// TIA Portal project "GestionCMD" (V17)

(* hardware
DEVICE "S7-1500/ET200MP station_1"  S7-1500 station
   slot 0: "Rail_0"  Rack  6ES7 590-1***0-0AA0
   slot 1: "PLC_1"  CPU 1516-3 PN/DP  6ES7 516-3AN02-0AB0  V2.9
      slot 3: "CPU display_1"  6ES7591-1BA00-0AA0
      slot 32768: "PROFINET interface_1"  X1
         slot 32769: "Port_1"  X1 P1
         slot 32770: "Port_2"  X1 P2
      slot 33024: "PROFINET interface_2"  X2
         slot 33025: "Port_1"  X2 P1
      slot 33280: "DP interface_1"  X3
      slot 34817: "Virtual CP interface port_1"  Virtual CP interface port  Virtual CP interface port
DEVICE "HMI_1"  KTP400 Comfort
   slot 0: "HMI_1"  KTP400 Comfort  6AV2 124-2DC01-0AX0  17.0.0.0
   slot 1: "HMI_RT_1"  KTP400 Comfort  6AV2 124-2DC01-0AX0  17.0.0.0
   slot 5: "HMI_1.IE_CP_1"  PROFINET Interface  17.0.0.0
      slot 1: "PROFINET Interface_1"  PROFINET Interface
         slot 1: "Port_1"  Port
   slot 7: "HMI_1.MPI/DP_CP_1"  MPI/DP Interface  17.0.0.0
*)

// ===== PLC "PLC_1"  CPU 1516-3 PN/DP =====

VAR_GLOBAL   // PLC tag table "Default tag table"
   "Etape1" AT %M0.0 : Bool;
   "Etape2" AT %M0.1 : Bool;
   "Etape3" AT %M0.2 : Bool;
   "MonterBarriere" AT %Q0.0 : Bool;
   "DescenteBarriere" AT %Q0.1 : Bool;
   "VoiturePasser" AT %M0.3 : Bool;
   "N_fois_badge" AT %MW10 : Int;
   "PositionBasBarriere" AT %M2.0 : Bool;
   "SignalBadge" AT %M2.1 : Bool;
   "Tag_1" AT %Q0.2 : Bool;
   "UpLevel" AT %I0.0 : Bool;
   "DownLevel" AT %I0.1 : Bool;
   "LevelFC" AT %MW30 : Int;
   "LevelFB" AT %MW34 : Int;
   "Tag_2" AT %M4.0 : Bool;
   "Tag_3" AT %M4.1 : Bool;
   "Tag_4" AT %M4.2 : Bool;
   "Tag_5" AT %M4.3 : Bool;
   "trigger" AT %M4.4 : Bool;
END_VAR

DATA_BLOCK "FB1"   // DB3
{ S7_Optimized_Access := 'TRUE' }
VERSION : 0.1
// stored: InstanceOfName Block_1
"Block_1"
BEGIN
END_DATA_BLOCK

DATA_BLOCK "FillingFB_DB"   // DB4
{ S7_Optimized_Access := 'TRUE' }
VERSION : 0.1
// stored: InstanceOfName FillingFB
"FillingFB"
BEGIN
END_DATA_BLOCK

FUNCTION_BLOCK "Block_1"   // FB1, SCL
{ S7_Optimized_Access := 'TRUE' }
VERSION : 0.1
   VAR
      MyNBBadge : Int;
   END_VAR
BEGIN
   IF "Etape1" AND "N_fois_badge" <> 0 THEN
       "Etape2" := TRUE;
       "Etape1" := FALSE;
   END_IF;

   IF "Etape2" AND "VoiturePasser" <> 0 THEN
       "Etape3" := TRUE;
       "Etape2" := FALSE;
   END_IF;

   IF "Etape3" AND "PositionBasBarriere" <> 0 THEN
       "Etape1" := TRUE;
       "Etape3" := FALSE;
   END_IF;

   "R_TRIG_DB"(CLK:="SignalBadge");
   "F_Etape1"(CLK := "Etape1");

   IF "R_TRIG_DB".Q THEN
       "N_fois_badge" += 1;
   END_IF;

   IF "F_Etape1".Q THEN
       "N_fois_badge" -= 1;
   END_IF;

   #MyNBBadge := "N_fois_badge";
END_FUNCTION_BLOCK

FUNCTION_BLOCK "FillingFB"   // FB2, LAD
{ S7_Optimized_Access := 'TRUE' }
VERSION : 0.1
   VAR_INPUT
      uplevel : Bool;
      downlevel : Bool;
   END_VAR
   VAR_OUTPUT
      OutLevel : Int;
   END_VAR
   VAR
      volum : Int;
   END_VAR
BEGIN

REGION Network 2
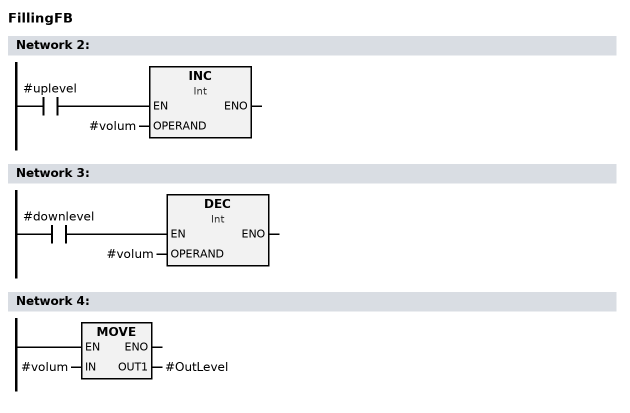
   RUNG wire#powerrail
      Contact( #uplevel )
      { S7_Templates := "DestType := Int" } Inc( #volum )
   END_RUNG
   // the same network as SCL:
   IF #uplevel THEN #volum := #volum + 1; END_IF;
END_REGION

REGION Network 3
   RUNG wire#powerrail
      Contact( #downlevel )
      { S7_Templates := "DestType := Int" } Dec( #volum )
   END_RUNG
   // the same network as SCL:
   IF #downlevel THEN #volum := #volum - 1; END_IF;
END_REGION

REGION Network 4
   RUNG wire#powerrail
      Move(in := #volum, out1 => #OutLevel)
   END_RUNG
   // the same network as SCL:
   #OutLevel := #volum;
END_REGION
END_FUNCTION_BLOCK

FUNCTION "FillingFC" : Void   // FC1, LAD
{ S7_Optimized_Access := 'TRUE' }
VERSION : 0.1
   VAR_INPUT
      uplevel : Bool;
      downlevel : Bool;
   END_VAR
   VAR_OUTPUT
      OutLevel : Int;
   END_VAR
   VAR_TEMP
      Volum : Int;
   END_VAR
   VAR CONSTANT
      Constant_1 : Int;
   END_VAR
BEGIN

REGION Network 1
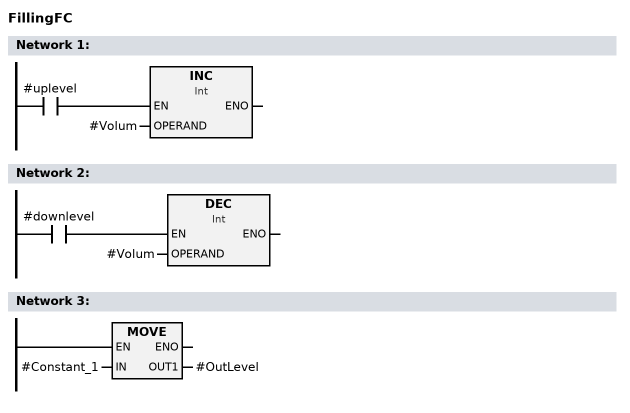
   RUNG wire#powerrail
      Contact( #uplevel )
      { S7_Templates := "DestType := Int" } Inc( #Volum )
   END_RUNG
   // the same network as SCL:
   IF #uplevel THEN #Volum := #Volum + 1; END_IF;
END_REGION

REGION Network 2
   RUNG wire#powerrail
      Contact( #downlevel )
      { S7_Templates := "DestType := Int" } Dec( #Volum )
   END_RUNG
   // the same network as SCL:
   IF #downlevel THEN #Volum := #Volum - 1; END_IF;
END_REGION

REGION Network 3
   RUNG wire#powerrail
      Move(in := #Constant_1, out1 => #OutLevel)
   END_RUNG
   // the same network as SCL:
   #OutLevel := #Constant_1;
END_REGION
END_FUNCTION

ORGANIZATION_BLOCK "Main"   // OB1, LAD, ProgramCycle
TITLE = "Main Program Sweep (Cycle)"
{ S7_Optimized_Access := 'TRUE' }
VERSION : 0.1
   VAR_INPUT
      Initial_Call : Bool;   // Initial call of this OB
      Remanence : Bool;   // =True, if remanent data are available
   END_VAR
   VAR_TEMP   // added for the SCL form of the ladder/FBD networks
      _w1 : Bool;
      _w2 : Bool;
   END_VAR
BEGIN

REGION Network 1
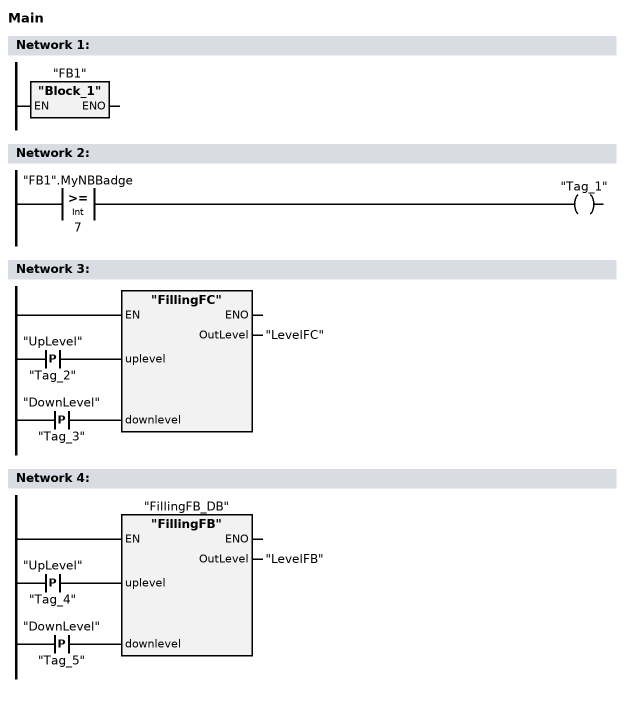
   RUNG wire#powerrail
      "FB1"()
   END_RUNG
   // the same network as SCL:
   "FB1"();   // "Block_1"
END_REGION

REGION Network 2
   RUNG wire#powerrail
      { S7_Templates := "SrcType := Int" } GE_Contact(in1 := "FB1".MyNBBadge, in2 := 7)
      Coil( "Tag_1" )
   END_RUNG
   // the same network as SCL:
   "Tag_1" := "FB1".MyNBBadge >= 7;
END_REGION

REGION Network 3
   RUNG wire#powerrail
      "FillingFC"(uplevel := wire#w1, downlevel := wire#w2, OutLevel => "LevelFC")
   END_RUNG
   RUNG wire#powerrail
      P_Contact(operand := "UpLevel", bit := "Tag_2")
   END_RUNG wire#w1
   RUNG wire#powerrail
      P_Contact(operand := "DownLevel", bit := "Tag_3")
   END_RUNG wire#w2
   // the same network as SCL:
   #_w1 := "UpLevel" AND NOT "Tag_2";   // rising edge of "UpLevel"
   "Tag_2" := "UpLevel";
   #_w2 := "DownLevel" AND NOT "Tag_3";   // rising edge of "DownLevel"
   "Tag_3" := "DownLevel";
   "FillingFC"(uplevel := #_w1, downlevel := #_w2, OutLevel => "LevelFC");
END_REGION

REGION Network 4
   RUNG wire#powerrail
      "FillingFB_DB"(uplevel := wire#w1, downlevel := wire#w2, OutLevel => "LevelFB")
   END_RUNG
   RUNG wire#powerrail
      P_Contact(operand := "UpLevel", bit := "Tag_4")
   END_RUNG wire#w1
   RUNG wire#powerrail
      P_Contact(operand := "DownLevel", bit := "Tag_5")
   END_RUNG wire#w2
   // the same network as SCL:
   #_w1 := "UpLevel" AND NOT "Tag_4";   // rising edge of "UpLevel"
   "Tag_4" := "UpLevel";
   #_w2 := "DownLevel" AND NOT "Tag_5";   // rising edge of "DownLevel"
   "Tag_5" := "DownLevel";
   "FillingFB_DB"(uplevel := #_w1, downlevel := #_w2, OutLevel => "LevelFB");   // "FillingFB"
END_REGION
END_ORGANIZATION_BLOCK

(* ===== HMI "HMI_RT_1" =====
system functions are stored by id; their names below are inferred from use
connection "HMI_Connection_1": ETHERNET, S7_1500_OMS

HMI tags "Default tag table"
   "Etape1" : Bool = PLC Etape1 AT %M0.0, 1 s
   "Etape2" : Bool = PLC Etape2 AT %M0.1, 1 s
   "Etape3" : Bool = PLC Etape3 AT %M0.2, 1 s
   "VoiturePasser" : Bool = PLC VoiturePasser AT %M0.3, 1 s
   "PositionBasBarriere" : Bool = PLC PositionBasBarriere AT %M2.0, 1 s
   "MonterBarriere" : Bool = PLC MonterBarriere AT %Q0.0, 1 s
   "DescenteBarriere" : Bool = PLC DescenteBarriere AT %Q0.1, 1 s
   "N_fois_badge" : Int = PLC N_fois_badge AT %MW10, 1 s
   "SignalBadge" : Bool = PLC SignalBadge AT %M2.1, 1 s
   "UpLevel" : Bool = PLC UpLevel AT %I0.0, 1 s
   "DownLevel" : Bool = PLC DownLevel AT %I0.1, 1 s
   "LevelFC" : Int = PLC LevelFC AT %MW30, 1 s
   "LevelFB" : Int = PLC LevelFB AT %MW34, 1 s
   "trigger" : Bool = PLC trigger AT %M4.4, 1 s

screen "Root screen" 480x272, template "Template_1"
   Button "Button_1" at 22,12 size 125x46; TextOff 'UP'
      on Press: function_b14e0dd5("UpLevel", 0)
   Button "Button_2" at 171,12 size 113x44; TextOff 'Down'
      on Press: function_b14e0dd5("DownLevel", 0)
   IOField "I/O field_3" at 357,162 size 96x32; FormatPattern s99999
      ProcessValue <- "LevelFC"
   IOField "I/O field_4" at 358,80 size 96x32; FormatPattern s99999
      ProcessValue <- "LevelFB"
   Button "Button_3" at 119,102 size 96x32; TextOff 'trigger'
      on Press: function_b14e0dd5("trigger", 0)
*)